PROGRAM P_FaultMonitoring
VAR_INPUT
		b_FaultReset: BOOL;
END_VAR


VAR

	n_Fault: ARRAY [0..1] OF DINT;
	b_FaultPending :BOOL;
	b_Faulted: BOOL;
	GlobalFaultTimer: ton; // all faults are checked in this interval.
	GlobalFaultTime: TIME:= T#1S;
	SR_0: SR;

	b_FaultImmediately: BOOL;

END_VAR
VAR // added by the converter: edge detectors and wires of the graphical bodies
    _rt1 : R_TRIG;
END_VAR

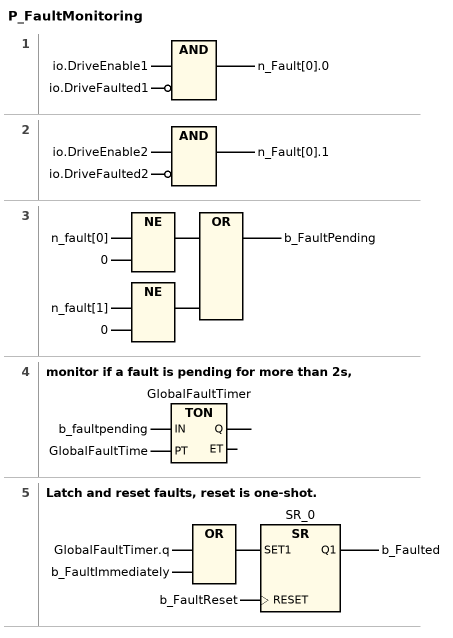
// NETWORK 1
n_Fault[0].0 := io.DriveEnable1 AND NOT io.DriveFaulted1;

// NETWORK 2
n_Fault[0].1 := io.DriveEnable2 AND NOT io.DriveFaulted2;

// NETWORK 3
b_FaultPending := n_fault[0] <> 0 OR n_fault[1] <> 0;

// NETWORK 4: monitor if a fault is pending for more than 2s,
GlobalFaultTimer(IN := b_faultpending, PT := GlobalFaultTime); // TON

// NETWORK 5: Latch and reset faults, reset is one-shot.
_rt1(CLK := b_FaultReset);
SR_0(SET1 := GlobalFaultTimer.q OR b_FaultImmediately, RESET := _rt1.Q); // SR
b_Faulted := SR_0.Q1;

END_PROGRAM

(* stored: Version 1.1.0.1, ProductVersion 3.1.4024.3
   POU P_FaultMonitoring: Id {810742e5-b0de-4c73-a054-43f34d3a704e}, SpecialFunc None *)
